// TIA Portal V19 export
DATA_BLOCK "Straightener_PERS"   // DB53
// stored: MemoryReserve 100
   VAR RETAIN
      PersistentValues : Struct
         Data : Struct
            Feed : "PositioningMachine_DataPers";
         END_STRUCT;
         Feed : "PositioningMachine_Par";
      END_STRUCT;
   END_VAR
BEGIN
   PersistentValues.Data.Feed.AxisEncoderSelection_OK := TRUE;
   PersistentValues.Data.Feed.AxisParameters_OK := TRUE;
   PersistentValues.Data.Feed.AxisReloadPostion_OK := TRUE;
   PersistentValues.Data.Feed.ActualPosition := 3798.845;
   PersistentValues.Feed.PosTolerance := 0.3;
   PersistentValues.Feed.DelayInPosition := T#300MS;
   PersistentValues.Feed.Man.VelBwd := 3000.0;
   PersistentValues.Feed.Man.VelFwdHigh := 3000.0;
   PersistentValues.Feed.Man.VelFwdLow := 3000.0;
   PersistentValues.Feed.Man.Acc := 500.0;
   PersistentValues.Feed.Man.Dec := 500.0;
   PersistentValues.Feed.Man.Jerk := 5000.0;
   PersistentValues.Feed.Man.DelayChangeVel := T#1MS;
   PersistentValues.Feed.Man.UsePositionControl := FALSE;
END_DATA_BLOCK
